// TIA Portal V19 export
FUNCTION_BLOCK "MainSafety"   // FB900, F_LAD
{ S7_Optimized_Access := 'TRUE' }
// stored: AutoNumber false
BEGIN

REGION Network 1: Read the safety data from Master PLC
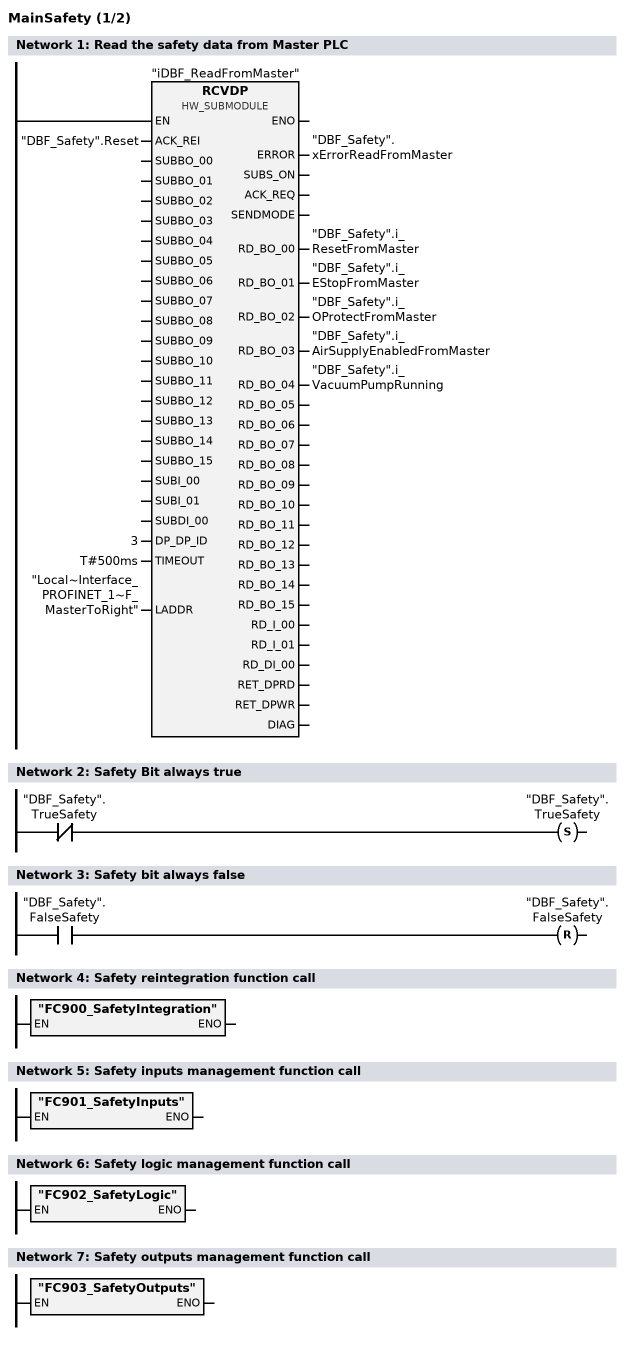
   RUNG wire#powerrail
      { S7_Templates := "laddr_type := HW_SUBMODULE" } "iDBF_ReadFromMaster".RCVDP(ACK_REI := "DBF_Safety".Reset, SUBBO_00 :=, SUBBO_01 :=, SUBBO_02 :=, SUBBO_03 :=, SUBBO_04 :=, SUBBO_05 :=, SUBBO_06 :=, SUBBO_07 :=, SUBBO_08 :=, SUBBO_09 :=, SUBBO_10 :=, SUBBO_11 :=, SUBBO_12 :=, SUBBO_13 :=, SUBBO_14 :=, SUBBO_15 :=, SUBI_00 :=, SUBI_01 :=, SUBDI_00 :=, DP_DP_ID := 3, TIMEOUT := T#500ms, LADDR := "Local~Interface_PROFINET_1~F_MasterToRight", ERROR => "DBF_Safety".xErrorReadFromMaster, SUBS_ON =>, ACK_REQ =>, SENDMODE =>, RD_BO_00 => "DBF_Safety".i_ResetFromMaster, RD_BO_01 => "DBF_Safety".i_EStopFromMaster, RD_BO_02 => "DBF_Safety".i_OProtectFromMaster, RD_BO_03 => "DBF_Safety".i_AirSupplyEnabledFromMaster, RD_BO_04 => "DBF_Safety".i_VacuumPumpRunning, RD_BO_05 =>, RD_BO_06 =>, RD_BO_07 =>, RD_BO_08 =>, RD_BO_09 =>, RD_BO_10 =>, RD_BO_11 =>, RD_BO_12 =>, RD_BO_13 =>, RD_BO_14 =>, RD_BO_15 =>, RD_I_00 =>, RD_I_01 =>, RD_DI_00 =>, RET_DPRD =>, RET_DPWR =>, DIAG =>)
   END_RUNG
   // the same network as SCL:
   "iDBF_ReadFromMaster"(ACK_REI := "DBF_Safety".Reset,   // RCVDP
                         DP_DP_ID := 3,
                         TIMEOUT := T#500ms,
                         LADDR := "Local~Interface_PROFINET_1~F_MasterToRight",
                         ERROR => "DBF_Safety".xErrorReadFromMaster,
                         RD_BO_00 => "DBF_Safety".i_ResetFromMaster,
                         RD_BO_01 => "DBF_Safety".i_EStopFromMaster,
                         RD_BO_02 => "DBF_Safety".i_OProtectFromMaster,
                         RD_BO_03 => "DBF_Safety".i_AirSupplyEnabledFromMaster,
                         RD_BO_04 => "DBF_Safety".i_VacuumPumpRunning);
END_REGION

REGION Network 2: Safety Bit always true
   RUNG wire#powerrail
      I_Contact( "DBF_Safety".TrueSafety )
      S_Coil( "DBF_Safety".TrueSafety )
   END_RUNG
   // the same network as SCL:
   IF NOT "DBF_Safety".TrueSafety THEN "DBF_Safety".TrueSafety := TRUE; END_IF;
END_REGION

REGION Network 3: Safety bit always false
   RUNG wire#powerrail
      Contact( "DBF_Safety".FalseSafety )
      R_Coil( "DBF_Safety".FalseSafety )
   END_RUNG
   // the same network as SCL:
   IF "DBF_Safety".FalseSafety THEN "DBF_Safety".FalseSafety := FALSE; END_IF;
END_REGION

REGION Network 4: Safety reintegration function call
   RUNG wire#powerrail
      "FC900_SafetyIntegration"()
   END_RUNG
   // the same network as SCL:
   "FC900_SafetyIntegration"();
END_REGION

REGION Network 5: Safety inputs management function call
   RUNG wire#powerrail
      "FC901_SafetyInputs"()
   END_RUNG
   // the same network as SCL:
   "FC901_SafetyInputs"();
END_REGION

REGION Network 6: Safety logic management function call
   RUNG wire#powerrail
      "FC902_SafetyLogic"()
   END_RUNG
   // the same network as SCL:
   "FC902_SafetyLogic"();
END_REGION

REGION Network 7: Safety outputs management function call
   RUNG wire#powerrail
      "FC903_SafetyOutputs"()
   END_RUNG
   // the same network as SCL:
   "FC903_SafetyOutputs"();
END_REGION

REGION Network 8: Write the safety data to Master PLC
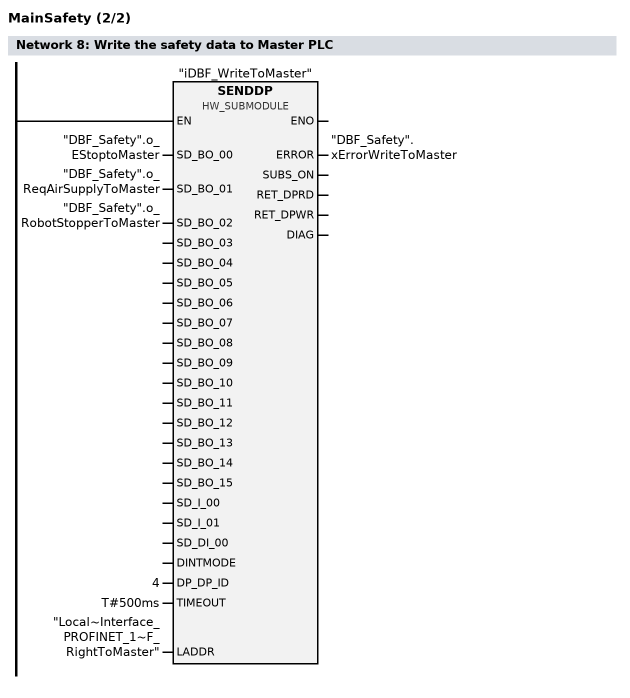
   RUNG wire#powerrail
      { S7_Templates := "laddr_type := HW_SUBMODULE" } "iDBF_WriteToMaster".SENDDP(SD_BO_00 := "DBF_Safety".o_EStoptoMaster, SD_BO_01 := "DBF_Safety".o_ReqAirSupplyToMaster, SD_BO_02 := "DBF_Safety".o_RobotStopperToMaster, SD_BO_03 :=, SD_BO_04 :=, SD_BO_05 :=, SD_BO_06 :=, SD_BO_07 :=, SD_BO_08 :=, SD_BO_09 :=, SD_BO_10 :=, SD_BO_11 :=, SD_BO_12 :=, SD_BO_13 :=, SD_BO_14 :=, SD_BO_15 :=, SD_I_00 :=, SD_I_01 :=, SD_DI_00 :=, DINTMODE :=, DP_DP_ID := 4, TIMEOUT := T#500ms, LADDR := "Local~Interface_PROFINET_1~F_RightToMaster", ERROR => "DBF_Safety".xErrorWriteToMaster, SUBS_ON =>, RET_DPRD =>, RET_DPWR =>, DIAG =>)
   END_RUNG
   // the same network as SCL:
   "iDBF_WriteToMaster"(SD_BO_00 := "DBF_Safety".o_EStoptoMaster,   // SENDDP
                        SD_BO_01 := "DBF_Safety".o_ReqAirSupplyToMaster,
                        SD_BO_02 := "DBF_Safety".o_RobotStopperToMaster,
                        DP_DP_ID := 4,
                        TIMEOUT := T#500ms,
                        LADDR := "Local~Interface_PROFINET_1~F_RightToMaster",
                        ERROR => "DBF_Safety".xErrorWriteToMaster);
END_REGION
END_FUNCTION_BLOCK
